(* IEC 61131-3 sources: RL_MAR/experiments/results/ablation/Ablation_no_role_config_deepseek-ai_DeepSeek-V3.2_20260603_074104 (part 2) *)

(* ---- med_49.st ---- *)
FUNCTION_BLOCK SmartHVACSystem
VAR_INPUT
    TemperatureSensor : REAL; (* Temperature sensor reading *)
    HumiditySensor : REAL; (* Humidity sensor reading *)
    Enable : BOOL := TRUE; (* System enable *)
    Reset : BOOL := FALSE; (* System reset *)
    ManualMode : BOOL := FALSE; (* Manual mode override *)
    ManualHVACMode : INT := 0; (* Manual HVAC mode: 0=Off, 1=Cooling, 2=Heating, 3=Ventilation *)
    ManualFanSpeed : INT := 0; (* Manual fan speed: 0=Off, 1=Low, 2=Medium, 3=High *)
END_VAR

VAR_OUTPUT
    HVACMode : INT := 0; (* HVAC operating mode: 0=Off, 1=Cooling, 2=Heating, 3=Ventilation *)
    HVACFanSpeed : INT := 0; (* Fan speed: 0=Off, 1=Low, 2=Medium, 3=High *)
    SystemActive : BOOL := FALSE; (* System active status *)
    Alarm : BOOL := FALSE; (* System alarm *)
END_VAR

VAR
    DesiredTemperature : REAL := 24.0; (* Desired temperature setting *)
    DesiredHumidity : REAL := 50.0; (* Desired humidity setting *)
    TemperatureThreshold : REAL := 1.0; (* Temperature tolerance threshold *)
    HumidityThreshold : REAL := 5.0; (* Humidity tolerance threshold *)

    AdjustedHumidity : REAL; (* Sanitized humidity input *)
    AdjustedTemperature : REAL; (* Sanitized temperature input *)

    NeedsVentilation : BOOL; (* Flag for ventilation requirement *)
    NeedsHeating : BOOL; (* Flag for heating requirement *)
    NeedsCooling : BOOL; (* Flag for cooling requirement *)

    TempSanitized : BOOL; (* Temperature sanitization status *)
    HumSanitized : BOOL; (* Humidity sanitization status *)

    ModeTimer : TON; (* Timer for mode changes *)
    FanTimer : TON; (* Timer for fan speed changes *)

    TempArray : ARRAY[1..10] OF REAL; (* Temperature history buffer *)
    HumArray : ARRAY[1..10] OF REAL; (* Humidity history buffer *)
    AvgTemperature : REAL; (* Average temperature *)
    AvgHumidity : REAL; (* Average humidity *)

    i : INT; (* Loop counter *)
    ArrayIndex : INT := 1; (* Current array index *)
    SampleCount : INT := 0; (* Number of samples collected *)
END_VAR

// Main execution logic
IF Reset THEN
    // Reset system
    HVACMode := 0;
    HVACFanSpeed := 0;
    SystemActive := FALSE;
    Alarm := FALSE;
    AdjustedHumidity := 0.0;
    AdjustedTemperature := 0.0;
    NeedsVentilation := FALSE;
    NeedsHeating := FALSE;
    NeedsCooling := FALSE;
    TempSanitized := FALSE;
    HumSanitized := FALSE;
    AvgTemperature := 0.0;
    AvgHumidity := 0.0;
    SampleCount := 0;
    ArrayIndex := 1;

    FOR i := 1 TO 10 DO
        TempArray[i] := 0.0;
        HumArray[i] := 0.0;
    END_FOR;

ELSIF Enable THEN
    SystemActive := TRUE;

    // 1. Input Sanitization
    // Sanitize humidity input
    IF HumiditySensor < 0.0 THEN
        AdjustedHumidity := 0.0;
        HumSanitized := TRUE;
    ELSIF HumiditySensor > 100.0 THEN
        AdjustedHumidity := 100.0;
        HumSanitized := TRUE;
    ELSE
        AdjustedHumidity := HumiditySensor;
        HumSanitized := TRUE;
    END_IF;

    // Sanitize temperature input
    IF TemperatureSensor < -50.0 THEN
        AdjustedTemperature := -50.0;
        TempSanitized := TRUE;
    ELSIF TemperatureSensor > 100.0 THEN
        AdjustedTemperature := 100.0;
        TempSanitized := TRUE;
    ELSE
        AdjustedTemperature := TemperatureSensor;
        TempSanitized := TRUE;
    END_IF;

    // Check for sensor alarm conditions
    Alarm := NOT (TempSanitized AND HumSanitized);

    // 2. Data averaging for stability
    TempArray[ArrayIndex] := AdjustedTemperature;
    HumArray[ArrayIndex] := AdjustedHumidity;

    ArrayIndex := ArrayIndex + 1;
    IF ArrayIndex > 10 THEN
        ArrayIndex := 1;
    END_IF;

    IF SampleCount < 10 THEN
        SampleCount := SampleCount + 1;
    END_IF;

    // Calculate averages
    AvgTemperature := 0.0;
    AvgHumidity := 0.0;
    FOR i := 1 TO SampleCount DO
        AvgTemperature := AvgTemperature + TempArray[i];
        AvgHumidity := AvgHumidity + HumArray[i];
    END_FOR;

    IF SampleCount > 0 THEN
        AvgTemperature := AvgTemperature / SampleCount;
        AvgHumidity := AvgHumidity / SampleCount;
    END_IF;

    // 3. Determine System Requirements using averaged values
    // Ventilation requirement
    IF AvgHumidity < (DesiredHumidity - HumidityThreshold) THEN
        NeedsVentilation := TRUE;
    ELSE
        NeedsVentilation := FALSE;
    END_IF;

    // Heating requirement
    IF AvgTemperature < (DesiredTemperature - TemperatureThreshold) THEN
        NeedsHeating := TRUE;
    ELSE
        NeedsHeating := FALSE;
    END_IF;

    // Cooling requirement
    IF AvgTemperature > (DesiredTemperature + TemperatureThreshold) THEN
        NeedsCooling := TRUE;
    ELSE
        NeedsCooling := FALSE;
    END_IF;

    // 4. Control Logic with prioritization
    IF ManualMode THEN
        // Manual mode override
        HVACMode := LIMIT(0, ManualHVACMode, 3);
        HVACFanSpeed := LIMIT(0, ManualFanSpeed, 3);
    ELSE
        // Automatic mode with prioritization
        IF NeedsHeating THEN
            HVACMode := 2; // Heating
            HVACFanSpeed := 3; // High
        ELSIF NeedsCooling THEN
            HVACMode := 1; // Cooling
            HVACFanSpeed := 3; // High
        ELSIF NeedsVentilation THEN
            HVACMode := 3; // Ventilation
            HVACFanSpeed := 3; // High
        ELSE
            HVACMode := 0; // Off
            HVACFanSpeed := 0; // Off
        END_IF;
    END_IF;

    // Apply timers for mode stability
    ModeTimer(IN := (HVACMode <> 0), PT := T#2S);
    FanTimer(IN := (HVACFanSpeed <> 0), PT := T#1S);

    // Ensure system only reports active when timers are done
    IF NOT ModeTimer.Q THEN
        HVACMode := 0;
    END_IF;

    IF NOT FanTimer.Q THEN
        HVACFanSpeed := 0;
    END_IF;

ELSE
    // System disabled
    SystemActive := FALSE;
    HVACMode := 0;
    HVACFanSpeed := 0;
    NeedsVentilation := FALSE;
    NeedsHeating := FALSE;
    NeedsCooling := FALSE;
END_IF;

END_FUNCTION_BLOCK

(* ---- med_50.st ---- *)
FUNCTION_BLOCK CarParkingSystem
VAR_INPUT
    NewCarSlot : INT; (* Input for new car arrival slot number *)
END_VAR
VAR_OUTPUT
    Elevator1Busy : BOOL; (* Elevator 1 status - busy or idle *)
    Elevator2Busy : BOOL; (* Elevator 2 status - busy or idle *)
    Elevator1Position : INT; (* Elevator 1 current position *)
    Elevator2Position : INT; (* Elevator 2 current position *)
END_VAR
VAR
    Elevator1Target : INT; (* Elevator 1 target floor *)
    Elevator2Target : INT; (* Elevator 2 target floor *)
    CarSlots : ARRAY[1..100] OF BOOL; (* Array to represent parking slots - TRUE if occupied *)
    bInitialized : BOOL := FALSE; (* Initialization flag *)
    i : INT; (* Loop index *)
    PendingRequests1 : ARRAY[1..50] OF BOOL; (* Pending requests for Elevator 1 *)
    PendingRequests2 : ARRAY[51..100] OF BOOL; (* Pending requests for Elevator 2 *)
    ScanIndex1 : INT := 1; (* Scanning index for Elevator 1 *)
    ScanIndex2 : INT := 51; (* Scanning index for Elevator 2 *)
END_VAR

(* Initialization - executed once *)
IF NOT bInitialized THEN
    Elevator1Busy := FALSE;
    Elevator2Busy := FALSE;
    Elevator1Position := 0;
    Elevator2Position := 0;
    Elevator1Target := 0;
    Elevator2Target := 0;

    (* Initialize all parking slots as empty *)
    FOR i := 1 TO 100 DO
        CarSlots[i] := FALSE;
    END_FOR;

    (* Initialize pending request arrays *)
    FOR i := 1 TO 50 DO
        PendingRequests1[i] := FALSE;
    END_FOR;

    FOR i := 51 TO 100 DO
        PendingRequests2[i] := FALSE;
    END_FOR;

    bInitialized := TRUE;
END_IF;

(* Process new car arrival if valid *)
IF (NewCarSlot >= 1) AND (NewCarSlot <= 100) THEN
    IF NOT CarSlots[NewCarSlot] THEN
        CarSlots[NewCarSlot] := TRUE;

        (* Store request in appropriate pending queue *)
        IF NewCarSlot <= 50 THEN
            PendingRequests1[NewCarSlot] := TRUE;
        ELSE
            PendingRequests2[NewCarSlot] := TRUE;
        END_IF;
    END_IF;
END_IF;

(* Control Elevator 1 movement *)
IF Elevator1Busy THEN
    IF Elevator1Position < Elevator1Target THEN
        Elevator1Position := Elevator1Position + 1;
    ELSIF Elevator1Position > Elevator1Target THEN
        Elevator1Position := Elevator1Position - 1;
    ELSE
        (* Elevator reached target - mark slot as serviced *)
        IF (Elevator1Target >= 1) AND (Elevator1Target <= 50) THEN
            PendingRequests1[Elevator1Target] := FALSE;
        END_IF;
        Elevator1Busy := FALSE;
    END_IF;
END_IF;

(* Control Elevator 2 movement *)
IF Elevator2Busy THEN
    IF Elevator2Position < Elevator2Target THEN
        Elevator2Position := Elevator2Position + 1;
    ELSIF Elevator2Position > Elevator2Target THEN
        Elevator2Position := Elevator2Position - 1;
    ELSE
        (* Elevator reached target - mark slot as serviced *)
        IF (Elevator2Target >= 51) AND (Elevator2Target <= 100) THEN
            PendingRequests2[Elevator2Target] := FALSE;
        END_IF;
        Elevator2Busy := FALSE;
    END_IF;
END_IF;

(* Idle elevator scanning for pending requests - Elevator 1 *)
IF NOT Elevator1Busy THEN
    (* Check for pending requests with round-robin scanning *)
    FOR i := 0 TO 49 DO
        ScanIndex1 := ScanIndex1 + 1;
        IF ScanIndex1 > 50 THEN
            ScanIndex1 := 1;
        END_IF;

        IF PendingRequests1[ScanIndex1] THEN
            Elevator1Target := ScanIndex1;
            Elevator1Busy := TRUE;
            EXIT;
        END_IF;
    END_FOR;
END_IF;

(* Idle elevator scanning for pending requests - Elevator 2 *)
IF NOT Elevator2Busy THEN
    (* Check for pending requests with round-robin scanning *)
    FOR i := 0 TO 49 DO
        ScanIndex2 := ScanIndex2 + 1;
        IF ScanIndex2 > 100 THEN
            ScanIndex2 := 51;
        END_IF;

        IF PendingRequests2[ScanIndex2] THEN
            Elevator2Target := ScanIndex2;
            Elevator2Busy := TRUE;
            EXIT;
        END_IF;
    END_FOR;
END_IF;

END_FUNCTION_BLOCK

(* ---- med_51.st ---- *)
FUNCTION_BLOCK PizzaMakingMachine
VAR_INPUT
    StartButton : BOOL;
    StopButton : BOOL;
    DoughReadySensor : BOOL;
    ToppingsReadySensor : BOOL;
    BakingDoneSensor : BOOL;
END_VAR

VAR_OUTPUT
    DoughRollerMotor : BOOL;
    ToppingDispenser : BOOL;
    ConveyorMotor : BOOL;
    OvenHeater : BOOL;
    OvenTemperature : INT;
END_VAR

VAR
    State : INT;
    OvenTargetTemp : INT;
END_VAR

// State definitions
CONSTANT
    STATE_IDLE : INT := 0;
    STATE_ROLLING_DOUGH : INT := 1;
    STATE_ADDING_TOPPINGS : INT := 2;
    STATE_MOVING_TO_OVEN : INT := 3;
    STATE_BAKING : INT := 4;
    STATE_COMPLETE : INT := 5;
END_CONSTANT

// Main state machine logic
IF StopButton THEN
    // Emergency stop - reset everything
    State := STATE_IDLE;
    DoughRollerMotor := FALSE;
    ToppingDispenser := FALSE;
    ConveyorMotor := FALSE;
    OvenHeater := FALSE;
    OvenTargetTemp := 0;
ELSE
    CASE State OF
        STATE_IDLE:
            DoughRollerMotor := FALSE;
            ToppingDispenser := FALSE;
            ConveyorMotor := FALSE;
            OvenHeater := FALSE;
            OvenTargetTemp := 0;

            IF StartButton THEN
                State := STATE_ROLLING_DOUGH;
            END_IF;

        STATE_ROLLING_DOUGH:
            DoughRollerMotor := TRUE;
            ToppingDispenser := FALSE;
            ConveyorMotor := FALSE;
            OvenHeater := FALSE;
            OvenTargetTemp := 0;

            IF DoughReadySensor THEN
                State := STATE_ADDING_TOPPINGS;
            END_IF;

        STATE_ADDING_TOPPINGS:
            DoughRollerMotor := FALSE;
            ToppingDispenser := TRUE;
            ConveyorMotor := FALSE;
            OvenHeater := FALSE;
            OvenTargetTemp := 0;

            IF ToppingsReadySensor THEN
                State := STATE_MOVING_TO_OVEN;
            END_IF;

        STATE_MOVING_TO_OVEN:
            DoughRollerMotor := FALSE;
            ToppingDispenser := FALSE;
            ConveyorMotor := TRUE;
            OvenHeater := TRUE; // Start heating oven
            OvenTargetTemp := 220;

            // Assume conveyor moves pizza to oven automatically
            // In real system, would have position sensor
            State := STATE_BAKING;

        STATE_BAKING:
            DoughRollerMotor := FALSE;
            ToppingDispenser := FALSE;
            ConveyorMotor := FALSE;
            OvenHeater := TRUE;
            OvenTargetTemp := 220;

            IF BakingDoneSensor THEN
                State := STATE_COMPLETE;
            END_IF;

        STATE_COMPLETE:
            DoughRollerMotor := FALSE;
            ToppingDispenser := FALSE;
            ConveyorMotor := FALSE;
            OvenHeater := FALSE;
            OvenTargetTemp := 0;

            // Wait for next start command
            IF NOT StartButton THEN
                State := STATE_IDLE;
            END_IF;

    END_CASE;
END_IF;

// Set oven temperature output
OvenTemperature := OvenTargetTemp;

END_FUNCTION_BLOCK

(* ---- med_52.st ---- *)
FUNCTION_BLOCK TrafficManagementSystem
VAR_INPUT
    VehicleCount1 : INT;
    VehicleCount2 : INT;
    VehicleCount3 : INT;
    VehicleCount4 : INT;
END_VAR

VAR_OUTPUT
    TrafficLight1 : BOOL;  (* TRUE = Green, FALSE = Red *)
    TrafficLight2 : BOOL;
    TrafficLight3 : BOOL;
    TrafficLight4 : BOOL;
END_VAR

VAR
    // Internal state variables for tie-breaking
    PrevPair1State : BOOL := TRUE;  (* Default to Intersection 1 green *)
    PrevPair2State : BOOL := TRUE;  (* Default to Intersection 3 green *)
END_VAR

(* Pair 1: Intersection 1 vs Intersection 2 *)
IF VehicleCount1 > VehicleCount2 THEN
    TrafficLight1 := TRUE;
    TrafficLight2 := FALSE;
    PrevPair1State := TRUE;
ELSIF VehicleCount2 > VehicleCount1 THEN
    TrafficLight1 := FALSE;
    TrafficLight2 := TRUE;
    PrevPair1State := FALSE;
ELSE
    (* Equal counts: use previous state to maintain complementary lights *)
    TrafficLight1 := PrevPair1State;
    TrafficLight2 := NOT PrevPair1State;
END_IF;

(* Pair 2: Intersection 3 vs Intersection 4 *)
IF VehicleCount3 > VehicleCount4 THEN
    TrafficLight3 := TRUE;
    TrafficLight4 := FALSE;
    PrevPair2State := TRUE;
ELSIF VehicleCount4 > VehicleCount3 THEN
    TrafficLight3 := FALSE;
    TrafficLight4 := TRUE;
    PrevPair2State := FALSE;
ELSE
    (* Equal counts: use previous state to maintain complementary lights *)
    TrafficLight3 := PrevPair2State;
    TrafficLight4 := NOT PrevPair2State;
END_IF;

END_FUNCTION_BLOCK

(* ---- med_53.st ---- *)
FUNCTION_BLOCK PouchMachine
VAR_INPUT
    start_machine: BOOL;
    stop_machine: BOOL;
END_VAR

VAR_OUTPUT
    machine_ready: BOOL;
    feeder_running: BOOL;
    cutter_running: BOOL;
    heating_running: BOOL;
    cooling_running: BOOL;
END_VAR

VAR
    startup_complete: BOOL := FALSE;
    shutdown_complete: BOOL := FALSE;
    current_state: INT := 0;
    next_state: INT := 0;

    // Timers for state transitions
    heating_timer: TON;
    cooling_timer: TON;
    feeder_timer: TON;
    cutter_timer: TON;

    // Additional internal variables
    tension_established: BOOL;
    heating_stations_active: ARRAY[1..8] OF BOOL;
    cooling_stations_active: ARRAY[1..8] OF BOOL;
    horizontal_cutter_active: BOOL;
    vertical_cutter_active: BOOL;
    feeder1_active: BOOL;
    feeder2_active: BOOL;

    // Loop counter
    i: INT;
END_VAR

// Initialize timers with preset times
heating_timer(IN := FALSE, PT := T#2S);
cooling_timer(IN := FALSE, PT := T#2S);
feeder_timer(IN := FALSE, PT := T#3S);
cutter_timer(IN := FALSE, PT := T#1S);

CASE current_state OF
    0: (* Idle State *)
        machine_ready := FALSE;
        feeder_running := FALSE;
        cutter_running := FALSE;
        heating_running := FALSE;
        cooling_running := FALSE;
        startup_complete := FALSE;
        shutdown_complete := FALSE;
        tension_established := FALSE;

        // Reset all stations
        FOR i := 1 TO 8 DO
            heating_stations_active[i] := FALSE;
            cooling_stations_active[i] := FALSE;
        END_FOR;

        horizontal_cutter_active := FALSE;
        vertical_cutter_active := FALSE;
        feeder1_active := FALSE;
        feeder2_active := FALSE;

        // Reset all timers
        heating_timer(IN := FALSE);
        cooling_timer(IN := FALSE);
        feeder_timer(IN := FALSE);
        cutter_timer(IN := FALSE);

        // Transition to start sequence
        IF start_machine AND NOT stop_machine THEN
            next_state := 1;
        ELSE
            next_state := 0;
        END_IF;

    1: (* Start Heating Stations *)
        heating_running := TRUE;

        // Activate all 8 heating stations
        FOR i := 1 TO 8 DO
            heating_stations_active[i] := TRUE;
        END_FOR;

        // Start timer for heating stabilization
        heating_timer(IN := TRUE);
        IF heating_timer.Q THEN
            next_state := 2;
            heating_timer(IN := FALSE);
        ELSE
            next_state := 1;
        END_IF;

    2: (* Start Cooling Stations *)
        cooling_running := TRUE;

        // Activate all 8 cooling stations
        FOR i := 1 TO 8 DO
            cooling_stations_active[i] := TRUE;
        END_FOR;

        // Start timer for cooling stabilization
        cooling_timer(IN := TRUE);
        IF cooling_timer.Q THEN
            next_state := 3;
            cooling_timer(IN := FALSE);
        ELSE
            next_state := 2;
        END_IF;

    3: (* Start Feeders with Tension Control *)
        feeder_running := TRUE;
        feeder1_active := TRUE;
        feeder2_active := TRUE;

        // Start timer for tension establishment
        feeder_timer(IN := TRUE);
        IF feeder_timer.Q THEN
            // Tension established after timer expires
            tension_established := TRUE;
            next_state := 4;
            feeder_timer(IN := FALSE);
        ELSE
            tension_established := FALSE;
            next_state := 3;
        END_IF;

    4: (* Start Cutters *)
        cutter_running := TRUE;
        horizontal_cutter_active := TRUE;
        vertical_cutter_active := TRUE;

        // Start timer for cutter activation
        cutter_timer(IN := TRUE);
        IF cutter_timer.Q THEN
            next_state := 5;
            cutter_timer(IN := FALSE);
        ELSE
            next_state := 4;
        END_IF;

    5: (* Machine Ready *)
        machine_ready := TRUE;
        startup_complete := TRUE;

        // Wait for stop command
        IF stop_machine THEN
            next_state := 6;
        ELSE
            next_state := 5;
        END_IF;

    6: (* Stop Cutters *)
        cutter_running := FALSE;
        horizontal_cutter_active := FALSE;
        vertical_cutter_active := FALSE;

        // Start timer for cutter deactivation
        cutter_timer(IN := TRUE);
        IF cutter_timer.Q THEN
            next_state := 7;
            cutter_timer(IN := FALSE);
        ELSE
            next_state := 6;
        END_IF;

    7: (* Stop Feeders *)
        feeder_running := FALSE;
        feeder1_active := FALSE;
        feeder2_active := FALSE;
        tension_established := FALSE;

        // Start timer for feeder shutdown
        feeder_timer(IN := TRUE);
        IF feeder_timer.Q THEN
            next_state := 8;
            feeder_timer(IN := FALSE);
        ELSE
            next_state := 7;
        END_IF;

    8: (* Stop Cooling Stations *)
        cooling_running := FALSE;

        // Deactivate all 8 cooling stations
        FOR i := 1 TO 8 DO
            cooling_stations_active[i] := FALSE;
        END_FOR;

        // Start timer for cooling shutdown
        cooling_timer(IN := TRUE);
        IF cooling_timer.Q THEN
            next_state := 9;
            cooling_timer(IN := FALSE);
        ELSE
            next_state := 8;
        END_IF;

    9: (* Stop Heating Stations *)
        heating_running := FALSE;

        // Deactivate all 8 heating stations
        FOR i := 1 TO 8 DO
            heating_stations_active[i] := FALSE;
        END_FOR;

        // Start timer for heating shutdown
        heating_timer(IN := TRUE);
        IF heating_timer.Q THEN
            next_state := 10;
            heating_timer(IN := FALSE);
        ELSE
            next_state := 9;
        END_IF;

    10: (* Shutdown Complete *)
        machine_ready := FALSE;
        shutdown_complete := TRUE;

        // Return to idle when stop signal is released
        IF NOT stop_machine THEN
            next_state := 0;
        ELSE
            next_state := 10;
        END_IF;

    ELSE
        // Safety fallback to idle state
        next_state := 0;
END_CASE;

// Update state for next scan cycle
current_state := next_state;

END_FUNCTION_BLOCK

(* ---- med_54.st ---- *)
FUNCTION_BLOCK FeedForwardControl
VAR_INPUT
    FlowRate1, FlowRate2: REAL; // Input flow rates of reactants
    MixRatio: REAL; // Desired mixing ratio (Reactant1:Reactant2)
END_VAR

VAR_OUTPUT
    OutFlowRate1, OutFlowRate2: REAL; // Output flow rates for reactants to maintain the mixing ratio
END_VAR

VAR
    MixedFlowRate: REAL; // Total mixed flow rate
    TempFlowRate1: REAL;
    TempFlowRate2: REAL;
    LimitedFlowRate1: REAL;
    LimitedFlowRate2: REAL;
END_VAR

// 1. VALIDATE AND LIMIT INPUT FLOW RATES (0 to 100)
IF FlowRate1 < 0.0 THEN
    LimitedFlowRate1 := 0.0;
ELSIF FlowRate1 > 100.0 THEN
    LimitedFlowRate1 := 100.0;
ELSE
    LimitedFlowRate1 := FlowRate1;
END_IF;

IF FlowRate2 < 0.0 THEN
    LimitedFlowRate2 := 0.0;
ELSIF FlowRate2 > 100.0 THEN
    LimitedFlowRate2 := 100.0;
ELSE
    LimitedFlowRate2 := FlowRate2;
END_IF;

// 2. CALCULATE TOTAL MIXED FLOW RATE
MixedFlowRate := LimitedFlowRate1 + LimitedFlowRate2;

// 3. CALCULATE OUTPUT FLOW RATES WITH ERROR HANDLING
IF MixRatio = 0.0 THEN
    // Prevent division by zero - use equal distribution
    TempFlowRate1 := MixedFlowRate / 2.0;
    TempFlowRate2 := MixedFlowRate / 2.0;
ELSE
    // Calculate based on mixing ratio: MixRatio = Reactant1:Reactant2
    // For ratio a:b, Reactant1 fraction = a/(a+b)
    TempFlowRate1 := MixedFlowRate * (MixRatio / (MixRatio + 1.0));
    TempFlowRate2 := MixedFlowRate * (1.0 / (MixRatio + 1.0));
END_IF;

// 4. LIMIT OUTPUT FLOW RATES TO ALLOWED RANGE (0 to 100)
IF TempFlowRate1 < 0.0 THEN
    OutFlowRate1 := 0.0;
ELSIF TempFlowRate1 > 100.0 THEN
    OutFlowRate1 := 100.0;
ELSE
    OutFlowRate1 := TempFlowRate1;
END_IF;

IF TempFlowRate2 < 0.0 THEN
    OutFlowRate2 := 0.0;
ELSIF TempFlowRate2 > 100.0 THEN
    OutFlowRate2 := 100.0;
ELSE
    OutFlowRate2 := TempFlowRate2;
END_IF;

// 5. ENSURE OUTPUT CONSISTENCY (Optional safeguard)
// Additional check to ensure outputs don't exceed total mixed flow rate
IF (OutFlowRate1 + OutFlowRate2) > MixedFlowRate THEN
    // Scale down proportionally if needed
    TempFlowRate1 := OutFlowRate1;
    TempFlowRate2 := OutFlowRate2;
    OutFlowRate1 := TempFlowRate1 * (MixedFlowRate / (TempFlowRate1 + TempFlowRate2));
    OutFlowRate2 := TempFlowRate2 * (MixedFlowRate / (TempFlowRate1 + TempFlowRate2));
END_IF;

END_FUNCTION_BLOCK

(* ---- med_55.st ---- *)
FUNCTION_BLOCK StateMachineControl
VAR_INPUT
    request : BOOL;
    done : BOOL;
END_VAR

VAR_OUTPUT
    listen : BOOL;
END_VAR

VAR
    state : INT := 0;
END_VAR

(* State machine logic *)
CASE state OF
    0: (* Idle state *)
        listen := TRUE;
        IF request THEN
            state := 1; (* Transition to Processing *)
            listen := FALSE;
        END_IF;

    1: (* Processing state *)
        listen := FALSE;
        IF done THEN
            state := 0; (* Transition to Idle *)
        END_IF;

    ELSE
        (* Error recovery - reset to Idle state *)
        state := 0;
        listen := TRUE;
END_CASE;

END_FUNCTION_BLOCK

(* ---- med_56.st ---- *)
FUNCTION_BLOCK FB_SimpleRepeat
VAR_INPUT
    INPUT_VAR1 : INT := 2;
    INPUT_COUNTER : INT := 4;
END_VAR

VAR_OUTPUT
    OUTPUT_VAR1 : INT;
END_VAR

VAR
    COUNTER : INT;
END_VAR

METHOD Main : BOOL
VAR_INPUT
    Execute : BOOL;
END_VAR
VAR_OUTPUT
    Done : BOOL;
END_VAR

    IF Execute THEN
        OUTPUT_VAR1 := INPUT_VAR1;
        COUNTER := INPUT_COUNTER;

        REPEAT
            OUTPUT_VAR1 := OUTPUT_VAR1 * 2;
            COUNTER := COUNTER - 1;
        UNTIL COUNTER <= 0
        END_REPEAT;

        Done := TRUE;
    ELSE
        Done := FALSE;
    END_IF;

    Main := Done;
END_METHOD

END_FUNCTION_BLOCK

(* ---- med_57.st ---- *)
FUNCTION_BLOCK FB_CourseDifferenceControl
VAR_INPUT
    KOMPASS_GRAD : INT;
    KURS : INT;
END_VAR
VAR_OUTPUT
    KURS_DIFF : INT;
END_VAR
VAR
    diff_temp : INT;
END_VAR

// Main logic
IF KOMPASS_GRAD < 0 THEN
    KURS_DIFF := 0;
ELSE
    diff_temp := KURS - KOMPASS_GRAD;

    // Apply range correction for angles
    IF diff_temp > 1800 THEN
        diff_temp := diff_temp - 3600;
    ELSIF diff_temp < -1800 THEN
        diff_temp := diff_temp + 3600;
    END_IF;

    KURS_DIFF := diff_temp;
END_IF;
END_FUNCTION_BLOCK

PROGRAM MAIN
VAR
    fbCourseDiff : FB_CourseDifferenceControl;
    kompass_grad_input : INT;
    kurs_input : INT;
    kurs_diff_output : INT;
END_VAR

// Call the function block
fbCourseDiff(KOMPASS_GRAD := kompass_grad_input, KURS := kurs_input);
kurs_diff_output := fbCourseDiff.KURS_DIFF;
END_PROGRAM

(* ---- med_58.st ---- *)
FUNCTION_BLOCK FB_ThresholdAccumulator
VAR_INPUT
    i : INT;
END_VAR

VAR_OUTPUT
    o : INT;
END_VAR

VAR
    s1 : INT;
END_VAR

// Initialize s1 to 0 at the start of each function block call
s1 := 0;

// If the input i is greater than 0, add its value to s1
IF i > 0 THEN
    s1 := s1 + i;
END_IF;

// After the first condition, if s1 equals 42, add 8000 to s1
IF s1 = 42 THEN
    s1 := s1 + 8000;
END_IF;

// Determine final output
IF s1 < 0 THEN
    o := 0;
ELSE
    o := s1;
END_IF;

END_FUNCTION_BLOCK

(* ---- med_59.st ---- *)
FUNCTION_BLOCK FB_ConditionalSelectAndAggregate
VAR_INPUT
    Z : INT;
END_VAR
VAR
    A_X : INT := 42;
    A_Y : INT := 333;
END_VAR
VAR_OUTPUT
    NEW_Z : INT;
END_VAR

IF A_X > Z THEN
    NEW_Z := A_Y;
ELSE
    NEW_Z := Z;
END_IF;
NEW_Z := NEW_Z + A_X + A_Y;
END_FUNCTION_BLOCK

(* ---- med_60.st ---- *)
FUNCTION_BLOCK FB_RequestHandler
VAR_INPUT
    request : BOOL;
    done : BOOL;
END_VAR

VAR_OUTPUT
    listen : BOOL;
END_VAR

VAR
    currentState : INT := 0;
    nextState : INT := 0;
END_VAR

CASE currentState OF
    0: (* State 0 - Idle/Listening *)
        listen := TRUE;

        IF request THEN
            listen := FALSE;
            nextState := 1;
        ELSE
            nextState := 0;
        END_IF;

    1: (* State 1 - Processing *)
        listen := FALSE;

        IF done THEN
            listen := TRUE;
            nextState := 0;
        ELSE
            nextState := 1;
        END_IF;

    ELSE
        (* Default case - return to state 0 if invalid state *)
        currentState := 0;
        nextState := 0;
        listen := TRUE;
END_CASE;

currentState := nextState;
END_FUNCTION_BLOCK

(* ---- med_61.st ---- *)
FUNCTION_BLOCK FB_Sum
VAR_INPUT
    maxValue : INT;
END_VAR
VAR_OUTPUT
    wData : WORD;
END_VAR
VAR
    II : INT;
    tempSum : DINT;
END_VAR

tempSum := 0;
FOR II := 0 TO maxValue DO
    tempSum := tempSum + II;
END_FOR;
wData := WORD(tempSum);
END_FUNCTION_BLOCK

(* ---- med_62.st ---- *)
FUNCTION_BLOCK FB_PedestrianTrafficLight
VAR_INPUT
    pedBtnPress : BOOL;
END_VAR
VAR_OUTPUT
    carLightIsGreen : BOOL;
    pedLightIsGreen : BOOL;
    counter : INT;
END_VAR
VAR
    buttonPressedBefore : BOOL := FALSE;
    state : INT := 1; // 1: Normal, 2: Wait for ped green, 3: Ped green, 4: Wait for car green
END_VAR

// State machine logic
CASE state OF
    1: // Normal state - Car green, Ped red
        carLightIsGreen := TRUE;
        pedLightIsGreen := FALSE;
        counter := 0;

        // Detect rising edge of button press
        IF pedBtnPress AND NOT buttonPressedBefore THEN
            state := 2;
        END_IF;

    2: // Car red, waiting for pedestrian green
        carLightIsGreen := FALSE;
        pedLightIsGreen := FALSE;
        counter := counter + 1;

        IF counter >= 10 THEN
            state := 3;
        END_IF;

    3: // Car red, pedestrian green
        carLightIsGreen := FALSE;
        pedLightIsGreen := TRUE;
        counter := counter + 1;

        IF counter >= 40 THEN
            state := 4;
        END_IF;

    4: // Car red, waiting for car green
        carLightIsGreen := FALSE;
        pedLightIsGreen := FALSE;
        counter := counter + 1;

        IF counter >= 50 THEN
            state := 1;
        END_IF;
END_CASE;

// Update button press tracking
buttonPressedBefore := pedBtnPress;

END_FUNCTION_BLOCK

(* ---- med_63.st ---- *)
FUNCTION MoveCarToExitGate : BOOL
VAR_INPUT
    SpaceNumber : INT;
END_VAR
// Car movement logic implementation
// Return TRUE when movement is successfully completed
MoveCarToExitGate := TRUE;
END_FUNCTION

FUNCTION_BLOCK Automated_Parking_Controller
VAR_INPUT
    EntryGateSensor : BOOL; (* Sensor input for entry gate *)
    ExitGateSensor : BOOL; (* Sensor input for exit gate *)
    CarDetected : BOOL; (* Sensor input for car detection *)
END_VAR
VAR_OUTPUT
    ParkingSpaceNumber : INT := 0; (* Allocated parking space number *)
    RetrievalInProgress : BOOL := FALSE; (* Flag for car retrieval in progress *)
END_VAR
VAR
    ParkingSpaces : ARRAY[1..100] OF BOOL; (* Parking space status: TRUE=Occupied, FALSE=Available *)
    i : INT; (* Loop counter *)
    AssignedSpace : INT := 0; (* Temporary storage for assigned space *)
    RetrievalComplete : BOOL := FALSE; (* Flag to track retrieval completion *)
END_VAR

// Entry Gate Management
IF EntryGateSensor AND NOT RetrievalInProgress THEN
    // Find first available parking space
    AssignedSpace := 0;
    FOR i := 1 TO 100 DO
        IF NOT ParkingSpaces[i] AND AssignedSpace = 0 THEN
            ParkingSpaces[i] := TRUE; // Mark as occupied
            ParkingSpaceNumber := i; // Output assigned space number
            AssignedSpace := i;
        END_IF
    END_FOR;
END_IF;

// Exit Gate Management
IF ExitGateSensor AND ParkingSpaceNumber > 0 THEN
    // Mark the corresponding parking space as available
    ParkingSpaces[ParkingSpaceNumber] := FALSE;
    ParkingSpaceNumber := 0; // Reset output
END_IF;

// Car Retrieval Management
IF CarDetected AND NOT RetrievalInProgress AND ParkingSpaceNumber > 0 THEN
    RetrievalInProgress := TRUE;
    RetrievalComplete := FALSE;
END_IF;

IF RetrievalInProgress THEN
    // Execute retrieval logic
    RetrievalComplete := MoveCarToExitGate(ParkingSpaceNumber);

    IF RetrievalComplete THEN
        // Mark parking space as available
        ParkingSpaces[ParkingSpaceNumber] := FALSE;
        ParkingSpaceNumber := 0; // Reset output
        RetrievalInProgress := FALSE; // Reset flag
    END_IF;
END_IF;
END_FUNCTION_BLOCK

(* ---- med_64.st ---- *)
FUNCTION_BLOCK BakeryOvenControl
VAR_INPUT
    TemperatureSensor : REAL;           (* Current oven temperature reading *)
    HumiditySensor : REAL;              (* Current oven humidity reading *)
    StartOven : BOOL;                   (* Command to start the oven *)
    TemperatureSetpoint : REAL;         (* Desired temperature setpoint *)
    HumiditySetpoint : REAL;            (* Desired humidity setpoint *)
    BakingTimeSetpoint : TIME;          (* Total baking time *)
    TemperatureThreshold : REAL := 2.0; (* Temperature control deadband *)
    HumidityThreshold : REAL := 5.0;    (* Humidity control deadband *)
END_VAR

VAR_OUTPUT
    HeatingElement : BOOL;              (* Control signal for heating element *)
    CoolingElement : BOOL;              (* Control signal for cooling element *)
    HumidityControl : BOOL;             (* Control signal for humidification *)
    DehumidityControl : BOOL;           (* Control signal for dehumidification *)
    OvenActive : BOOL;                  (* Oven status: TRUE when baking *)
    RemainingTime : TIME;               (* Remaining baking time *)
END_VAR

VAR
    BakingTimer : TON;                  (* Timer for baking duration *)
    OneSecondPulse : TON;               (* Timer for 1-second pulse generation *)
    PulseSignal : BOOL;                 (* Internal 1-second pulse *)
    InternalRemainingTime : TIME;       (* Internal remaining time counter *)
END_VAR

(* Initialize timers *)
OneSecondPulse(IN := NOT OneSecondPulse.Q, PT := T#1S);
PulseSignal := OneSecondPulse.Q;

(* Oven control logic *)
IF StartOven AND NOT OvenActive THEN
    (* Start baking cycle *)
    OvenActive := TRUE;
    InternalRemainingTime := BakingTimeSetpoint;
    BakingTimer(IN := TRUE, PT := BakingTimeSetpoint);
ELSIF NOT StartOven THEN
    (* Manual stop or initialization *)
    OvenActive := FALSE;
    BakingTimer(IN := FALSE, PT := T#0S);
END_IF

(* Decrement remaining time when oven is active *)
IF OvenActive AND PulseSignal THEN
    IF InternalRemainingTime >= T#1S THEN
        InternalRemainingTime := InternalRemainingTime - T#1S;
    ELSE
        InternalRemainingTime := T#0S;
    END_IF;
END_IF;

(* Stop oven when timer expires *)
IF BakingTimer.Q THEN
    OvenActive := FALSE;
END_IF;

(* Temperature control - only active when oven is on *)
IF OvenActive THEN
    HeatingElement := TemperatureSensor < (TemperatureSetpoint - TemperatureThreshold);
    CoolingElement := TemperatureSensor > (TemperatureSetpoint + TemperatureThreshold);
ELSE
    HeatingElement := FALSE;
    CoolingElement := FALSE;
END_IF;

(* Humidity control - only active when oven is on *)
IF OvenActive THEN
    HumidityControl := HumiditySensor < (HumiditySetpoint - HumidityThreshold);
    DehumidityControl := HumiditySensor > (HumiditySetpoint + HumidityThreshold);
ELSE
    HumidityControl := FALSE;
    DehumidityControl := FALSE;
END_IF;

(* Output remaining time *)
RemainingTime := InternalRemainingTime;

(* Ensure all outputs are off when oven is not active *)
IF NOT OvenActive THEN
    HeatingElement := FALSE;
    CoolingElement := FALSE;
    HumidityControl := FALSE;
    DehumidityControl := FALSE;
    InternalRemainingTime := T#0S;
END_IF;
END_FUNCTION_BLOCK

(* ---- med_65.st ---- *)
FUNCTION_BLOCK TheaterControl
VAR_INPUT
    StartButton : BOOL;        (* Input for starting a performance *)
    StopButton : BOOL;         (* Input for stopping a performance *)
    SceneNumber : INT;         (* Input for selecting the scene or act *)
END_VAR
VAR_OUTPUT
    LightingControl : BOOL;    (* Output for controlling lighting *)
    SoundControl : BOOL;       (* Output for controlling sound *)
    PerformanceInProgress : BOOL; (* Indicator for an ongoing performance *)
END_VAR
VAR
    bStartRisingEdge : BOOL;
    bStopRisingEdge : BOOL;
    bPrevStart : BOOL := FALSE;
    bPrevStop : BOOL := FALSE;
END_VAR

(* Detect rising edges for button presses *)
bStartRisingEdge := StartButton AND NOT bPrevStart;
bStopRisingEdge := StopButton AND NOT bPrevStop;
bPrevStart := StartButton;
bPrevStop := StopButton;

(* Main control logic with stop button having highest priority *)
IF bStopRisingEdge THEN
    (* Immediate stop - override all other inputs *)
    LightingControl := FALSE;
    SoundControl := FALSE;
    PerformanceInProgress := FALSE;
ELSIF bStartRisingEdge AND NOT PerformanceInProgress THEN
    (* Start performance only if not already in progress *)
    IF (SceneNumber >= 1) AND (SceneNumber <= 3) THEN
        (* Valid scene - activate outputs *)
        LightingControl := TRUE;
        SoundControl := TRUE;
        PerformanceInProgress := TRUE;
    ELSE
        (* Invalid scene - keep outputs inactive *)
        LightingControl := FALSE;
        SoundControl := FALSE;
        PerformanceInProgress := FALSE;
    END_IF;
END_IF;

(* Note: Outputs maintain their state until changed by the logic above *)
END_FUNCTION_BLOCK

(* ---- med_66.st ---- *)
FUNCTION_BLOCK ElevatorControl
VAR_INPUT
    CurrentPos : INT;
    RequestedPos : INT;
    ButtonPressed : BOOL;
END_VAR
VAR_OUTPUT
    MotorMovingUp : BOOL;
    MotorMovingDown : BOOL;
    DoorIsOpen : BOOL;
END_VAR
VAR
    bMoving : BOOL := FALSE;
END_VAR

// Main elevator control logic
IF ButtonPressed THEN
    // Start movement when button is pressed
    bMoving := TRUE;
    DoorIsOpen := FALSE;
END_IF;

IF bMoving THEN
    // Elevator is in motion
    IF RequestedPos > CurrentPos THEN
        // Move upward
        MotorMovingUp := TRUE;
        MotorMovingDown := FALSE;
        DoorIsOpen := FALSE;
    ELSIF RequestedPos < CurrentPos THEN
        // Move downward
        MotorMovingUp := FALSE;
        MotorMovingDown := TRUE;
        DoorIsOpen := FALSE;
    ELSE
        // Reached target floor
        MotorMovingUp := FALSE;
        MotorMovingDown := FALSE;
        DoorIsOpen := TRUE;
        bMoving := FALSE;
    END_IF;
ELSE
    // Elevator is stationary
    MotorMovingUp := FALSE;
    MotorMovingDown := FALSE;

    // Keep door open if at requested position, otherwise closed
    IF CurrentPos = RequestedPos THEN
        DoorIsOpen := TRUE;
    ELSE
        DoorIsOpen := FALSE;
    END_IF;
END_IF;

END_FUNCTION_BLOCK

(* ---- med_67.st ---- *)
FUNCTION_BLOCK FB_FactorialCalculator
VAR_INPUT
    X : INT;
END_VAR

VAR_OUTPUT
    FactorialResult : INT;
    FactorialGoodResult : INT;
END_VAR

VAR
END_VAR

// Initialize outputs
FactorialGoodResult := 0;
FactorialResult := 0;

// Check if input is within safe range
IF (X >= -3) AND (X <= 3) THEN
    // Calculate X^4 (X multiplied by itself 4 times)
    FactorialGoodResult := X * X * X * X;

    // Calculate FactorialResult based on FactorialGoodResult
    IF FactorialGoodResult > 1 THEN
        FactorialResult := FactorialGoodResult * (FactorialGoodResult - 1);
    ELSE
        FactorialResult := FactorialGoodResult;
    END_IF;
ELSE
    // Overflow prevention for inputs outside range
    FactorialResult := 1;
    FactorialGoodResult := 0;
END_IF;

END_FUNCTION_BLOCK

(* ---- med_68.st ---- *)
FUNCTION_BLOCK SignalControl
VAR_INPUT
    Int1 : BOOL;
    Int2 : BOOL;
    Int3 : BOOL;
    Int4 : BOOL;
    Int5 : BOOL;
    Int6 : BOOL;
    Int7 : BOOL;
    Int8 : BOOL;
    IntAn1 : UINT;
    IntAn2 : UINT;
    IntAn3 : UINT;
    IntAn4 : UINT;
    IntAn5 : UINT;
    IntAn6 : UINT;
    IntAn7 : UINT;
    IntAn8 : UINT;
    Marca2 : BOOL;
END_VAR

VAR_OUTPUT
    Out1 : BOOL;
    Out2 : BOOL;
    Out3 : BOOL;
    Out4 : BOOL;
    Out5 : BOOL;
    Out6 : BOOL;
    Out7 : BOOL;
    Out8 : BOOL;
    OutAn1 : UINT;
    OutAn2 : UINT;
    OutAn3 : UINT;
    OutAn4 : UINT;
    OutAn5 : UINT;
    OutAn6 : UINT;
    OutAn7 : UINT;
    OutAn8 : UINT;
END_VAR

VAR
    Marca1 : BOOL;
END_VAR

// Main logic execution
// Logic for Marca1 flag
IF NOT Marca2 AND (Marca1 OR NOT Out1) AND Int1 THEN
    Marca1 := TRUE;
ELSE
    Marca1 := FALSE;
END_IF;

// Logic for Marca2 flag (note: Marca2 is both input and internal state)
IF NOT Marca1 AND (Marca2 OR Out1) AND Int1 THEN
    Marca2 := TRUE;
ELSE
    Marca2 := FALSE;
END_IF;

// Latch behavior for Out1
IF NOT Marca2 AND (Marca1 OR Out1) THEN
    Out1 := TRUE;
ELSE
    Out1 := FALSE;
END_IF;

// Boolean pass-through for Out2, Out3, Out4
Out2 := Int2;
Out3 := Int3;
Out4 := Int4;

// Unsigned integer pass-through for OutAn1 to OutAn4
OutAn1 := IntAn1;
OutAn2 := IntAn2;
OutAn3 := IntAn3;
OutAn4 := IntAn4;

// Conditional output logic for Out5 to Out8
// Out5 condition: IntAn5 > 1000 AND NOT Int5
Out5 := (IntAn5 > 1000) AND NOT Int5;

// Out6 condition: IntAn6 > 1000 AND NOT Int6
Out6 := (IntAn6 > 1000) AND NOT Int6;

// Out7 condition: IntAn7 > 1000 AND NOT Int7
Out7 := (IntAn7 > 1000) AND NOT Int7;

// Out8 condition: IntAn8 > 1000 AND NOT Int8
Out8 := (IntAn8 > 1000) AND NOT Int8;

// Pass-through for analog outputs OutAn5 to OutAn8
OutAn5 := IntAn5;
OutAn6 := IntAn6;
OutAn7 := IntAn7;
OutAn8 := IntAn8;

END_FUNCTION_BLOCK

(* ---- med_69.st ---- *)
FUNCTION_BLOCK FB_ValueOut
VAR_INPUT
    valueIn : INT;
    conf : UINT;
END_VAR
VAR_OUTPUT
    ValueOut : INT;
END_VAR

CASE conf OF
    1,2:
        ValueOut := valueIn / 10;

    3:
        IF valueIn = 0 THEN
            ValueOut := 0;
        ELSIF valueIn = 300 THEN
            ValueOut := 163;
        ELSIF valueIn = 600 THEN
            ValueOut := 331;
        ELSE
            ValueOut := 0;
        END_IF;

    6,7:
        IF valueIn = 100 THEN
            ValueOut := 319;
        ELSE
            ValueOut := 0;
        END_IF;

    ELSE
        ValueOut := 0;
END_CASE;

END_FUNCTION_BLOCK

(* ---- med_70.st ---- *)
FUNCTION_BLOCK EggIncubatorControl
VAR_INPUT
    StartButton : BOOL;          (* Input for starting the incubation process *)
    StopButton : BOOL;           (* Input for stopping the incubation process *)
    TemperatureSensor : REAL;    (* Input for temperature reading in °C *)
    HumiditySensor : REAL;       (* Input for humidity reading in % *)
END_VAR
VAR_OUTPUT
    HeatingElement : BOOL;       (* Output for controlling the heating element *)
    Humidifier : BOOL;           (* Output for controlling the humidifier *)
    EggTurningMotor : BOOL;      (* Output for controlling the egg turning motor *)
    IncubationInProgress : BOOL; (* Indicator for an ongoing incubation process *)
END_VAR
VAR
    TargetTemperature : REAL;    (* Target temperature in °C *)
    TargetHumidity : REAL;       (* Target humidity in % *)
    TurnIntervalSeconds : INT;   (* Interval for turning eggs (1 hour in seconds) *)
    TurnTimerSeconds : INT;      (* Timer for egg turning cycle in seconds *)
END_VAR

(* Initialize control parameters *)
TargetTemperature := 37.5;
TargetHumidity := 50.0;
TurnIntervalSeconds := 3600;

(* Start/Stop Control *)
IF StopButton THEN
    IncubationInProgress := FALSE;
    HeatingElement := FALSE;
    Humidifier := FALSE;
    EggTurningMotor := FALSE;
    TurnTimerSeconds := 0;
ELSIF StartButton AND NOT IncubationInProgress THEN
    IncubationInProgress := TRUE;
END_IF;

(* Temperature Control *)
IF IncubationInProgress THEN
    IF TemperatureSensor < TargetTemperature THEN
        HeatingElement := TRUE;
    ELSE
        HeatingElement := FALSE;
    END_IF;
ELSE
    HeatingElement := FALSE;
END_IF;

(* Humidity Control *)
IF IncubationInProgress THEN
    IF HumiditySensor < TargetHumidity THEN
        Humidifier := TRUE;
    ELSE
        Humidifier := FALSE;
    END_IF;
ELSE
    Humidifier := FALSE;
END_IF;

(* Egg Turning Cycle *)
IF IncubationInProgress THEN
    TurnTimerSeconds := TurnTimerSeconds + 1;
    IF TurnTimerSeconds >= TurnIntervalSeconds THEN
        EggTurningMotor := NOT EggTurningMotor;
        TurnTimerSeconds := 0;
    END_IF;
ELSE
    TurnTimerSeconds := 0;
END_IF;

END_FUNCTION_BLOCK

(* ---- med_71.st ---- *)
FUNCTION_BLOCK FB_Fibonacci_Calculator
VAR_INPUT
    N : DINT := 5;
END_VAR
VAR_OUTPUT
    O : DINT := 1;
END_VAR
VAR
    F1 : DINT := 1;
    F2 : DINT := 1;
    CNT : DINT := 2;
    TempSum : DINT;
END_VAR

(* Handle edge cases: N <= 2 returns 1 *)
IF N <= 2 THEN
    O := 1;
ELSE
    (* Initialize Fibonacci sequence *)
    F1 := 1;
    F2 := 1;
    CNT := 2;

    (* Calculate Fibonacci numbers up to N-th term *)
    WHILE CNT < N DO
        TempSum := F1 + F2;

        (* Apply saturation arithmetic: clamp at INT maximum (32767) *)
        IF TempSum > 32767 THEN
            F2 := 32767;
            EXIT;  (* Exit loop early when saturation limit reached *)
        END_IF;

        (* Update Fibonacci values for next iteration *)
        F1 := F2;
        F2 := TempSum;
        CNT := CNT + 1;
    END_WHILE;

    (* Set output to the N-th Fibonacci number *)
    O := F2;
END_IF;
END_FUNCTION_BLOCK

(* ---- med_72.st ---- *)
FUNCTION_BLOCK DigitalSignageManagement
VAR_INPUT
    DisplayLocations : ARRAY[1..10] OF BOOL;    (* Display active status per location *)
    ContentSource : ARRAY[1..10] OF INT;        (* Requested content per location *)
END_VAR
VAR_OUTPUT
    CurrentContent : ARRAY[1..10] OF INT;       (* Actual displayed content per location *)
END_VAR
VAR
    i : INT;                                    (* Loop index *)
END_VAR

(* Process all 10 display locations *)
FOR i := 1 TO 10 DO
    IF DisplayLocations[i] THEN
        (* Display is active - validate content code *)
        CASE ContentSource[i] OF
            1: CurrentContent[i] := 1;          (* News *)
            2: CurrentContent[i] := 2;          (* Weather *)
            3: CurrentContent[i] := 3;          (* Promotional Content *)
        ELSE
            CurrentContent[i] := 0;             (* Invalid code - show no content *)
        END_CASE;
    ELSE
        (* Display is inactive - always show no content *)
        CurrentContent[i] := 0;
    END_IF;
END_FOR;

END_FUNCTION_BLOCK

(* ---- med_73.st ---- *)
FUNCTION_BLOCK RoboticWeldingSystem
VAR_INPUT
    RobotArm1Ready : BOOL;    (* Input for robot arm 1 ready status *)
    RobotArm2Ready : BOOL;    (* Input for robot arm 2 ready status *)
    WeldingGunReady : BOOL;   (* Input for welding gun ready status *)
    StartButton : BOOL;       (* Input for start button press *)
    StopButton : BOOL;        (* Input for stop button press *)
END_VAR
VAR_OUTPUT
    WeldingTrigger : BOOL;    (* Output to trigger welding *)
    WeldingComplete : BOOL;   (* Output indicating welding completion *)
END_VAR
VAR
    bAllReady : BOOL;         (* Internal flag for all components ready *)
END_VAR

(* Check if all components are ready *)
bAllReady := RobotArm1Ready AND RobotArm2Ready AND WeldingGunReady;

(* Main safety logic with stop button having highest priority *)
IF StopButton THEN
    (* Immediate stop when stop button is pressed *)
    WeldingTrigger := FALSE;
    WeldingComplete := TRUE;
ELSIF bAllReady AND StartButton THEN
    (* Start welding only when all components ready AND start button pressed *)
    WeldingTrigger := TRUE;
    WeldingComplete := FALSE;
ELSE
    (* Default state - no welding *)
    WeldingTrigger := FALSE;
    WeldingComplete := TRUE;
END_IF;

END_FUNCTION_BLOCK

(* ---- med_74.st ---- *)
FUNCTION_BLOCK TrafficManagementSystem
VAR_INPUT
    VehicleCount1 : INT; (* Vehicle count at intersection 1 *)
    VehicleCount2 : INT; (* Vehicle count at intersection 2 *)
    VehicleCount3 : INT; (* Vehicle count at intersection 3 *)
    VehicleCount4 : INT; (* Vehicle count at intersection 4 *)
END_VAR

VAR_OUTPUT
    TrafficLight1 : BOOL; (* TRUE = Green, FALSE = Red *)
    TrafficLight2 : BOOL; (* TRUE = Green, FALSE = Red *)
    TrafficLight3 : BOOL; (* TRUE = Green, FALSE = Red *)
    TrafficLight4 : BOOL; (* TRUE = Green, FALSE = Red *)
END_VAR

VAR
    (* Internal state variables for clarity *)
    TrafficLightState1 : BOOL;
    TrafficLightState2 : BOOL;
    TrafficLightState3 : BOOL;
    TrafficLightState4 : BOOL;
END_VAR

(* Control logic for intersection pair 1 (Intersection 1 and 2) *)
IF VehicleCount1 > VehicleCount2 THEN
    TrafficLightState1 := TRUE;   (* Green for intersection 1 *)
    TrafficLightState2 := FALSE;  (* Red for intersection 2 *)
ELSIF VehicleCount1 < VehicleCount2 THEN
    TrafficLightState1 := FALSE;  (* Red for intersection 1 *)
    TrafficLightState2 := TRUE;   (* Green for intersection 2 *)
ELSE
    (* Equal counts: both red for safety *)
    TrafficLightState1 := FALSE;
    TrafficLightState2 := FALSE;
END_IF;

(* Control logic for intersection pair 2 (Intersection 3 and 4) *)
IF VehicleCount3 > VehicleCount4 THEN
    TrafficLightState3 := TRUE;   (* Green for intersection 3 *)
    TrafficLightState4 := FALSE;  (* Red for intersection 4 *)
ELSIF VehicleCount3 < VehicleCount4 THEN
    TrafficLightState3 := FALSE;  (* Red for intersection 3 *)
    TrafficLightState4 := TRUE;   (* Green for intersection 4 *)
ELSE
    (* Equal counts: both red for safety *)
    TrafficLightState3 := FALSE;
    TrafficLightState4 := FALSE;
END_IF;

(* Assign internal states to outputs *)
TrafficLight1 := TrafficLightState1;
TrafficLight2 := TrafficLightState2;
TrafficLight3 := TrafficLightState3;
TrafficLight4 := TrafficLightState4;

END_FUNCTION_BLOCK

(* ---- med_75.st ---- *)
FUNCTION_BLOCK HomeBrewingSystem
VAR_INPUT
    TemperatureSensor : REAL; (* Input for temperature measurement (°C) *)
    WaterFlowSensor : REAL; (* Input for water flow measurement (L/min) *)
    BrewingStartTime : TIME; (* Input for brewing process start time *)
    BrewingDuration : TIME; (* Input for total brewing duration *)
END_VAR

VAR_OUTPUT
    HeatingElement : BOOL; (* Output to control heating element *)
    AgitationMotor : BOOL; (* Output to control agitation motor *)
    HopsDispenser : BOOL; (* Output to control hops dispenser *)
    FermentationTank : BOOL; (* Output to control fermentation tank *)
END_VAR

VAR
    ElapsedBrewingTime : TIME; (* Time elapsed since brewing start *)
    HopsDispensed : BOOL; (* Flag to track if hops have been dispensed *)
    TankTransferred : BOOL; (* Flag to track if transfer to fermentation tank has occurred *)
    CurrentTime : TIME; (* Current system time *)
    HopsTime : TIME := T#5h; (* Time threshold for hops dispensing *)
    FermentationTime : TIME := T#48h; (* Time threshold for fermentation transfer *)
    TargetTemperature : REAL := 65.0; (* Target brewing temperature *)
    FlowThreshold : REAL := 0.5; (* Flow threshold for agitation motor *)
END_VAR

(* Main program logic *)
CurrentTime := TIME(); (* Get current system time *)

(* Calculate elapsed brewing time *)
IF BrewingStartTime > T#0s THEN
    ElapsedBrewingTime := CurrentTime - BrewingStartTime;

    (* Ensure elapsed time doesn't exceed brewing duration *)
    IF ElapsedBrewingTime > BrewingDuration THEN
        ElapsedBrewingTime := BrewingDuration;
    END_IF;
ELSE
    ElapsedBrewingTime := T#0s;
END_IF;

(* Temperature control logic *)
HeatingElement := TemperatureSensor < TargetTemperature;

(* Agitation motor control logic *)
AgitationMotor := WaterFlowSensor > FlowThreshold;

(* Hops dispensing logic - activate after 5 hours, only once *)
IF (ElapsedBrewingTime >= HopsTime) AND (NOT HopsDispensed) AND (ElapsedBrewingTime <= BrewingDuration) THEN
    HopsDispenser := TRUE;
    HopsDispensed := TRUE;
ELSE
    HopsDispenser := FALSE;
END_IF;

(* Fermentation tank transfer logic - activate after 48 hours, only once *)
IF (ElapsedBrewingTime >= FermentationTime) AND (NOT TankTransferred) AND (ElapsedBrewingTime <= BrewingDuration) THEN
    FermentationTank := TRUE;
    TankTransferred := TRUE;
ELSE
    FermentationTank := FALSE;
END_IF;

(* Reset flags when brewing duration is complete or not started *)
IF (ElapsedBrewingTime >= BrewingDuration) OR (BrewingStartTime = T#0s) THEN
    HopsDispensed := FALSE;
    TankTransferred := FALSE;
END_IF;

END_FUNCTION_BLOCK

(* ---- med_76.st ---- *)
FUNCTION_BLOCK MultimediaArtInstallationControl
VAR_INPUT
    MotionSensor : BOOL;           (* Motion detection input *)
    AudioTrack : BOOL;             (* Selected audio track *)
    VisualContent : BOOL;          (* Selected visual content *)
END_VAR

VAR_OUTPUT
    LightingControl : BOOL;        (* Lighting control output *)
    AudioControl : BOOL;           (* Audio playback control *)
    VisualControl : BOOL;          (* Visual display control *)
    ActivationTime : TIME;         (* Activation duration *)
END_VAR

VAR
    ActivationTimer : TON;         (* Timer for activation duration *)
    TimerPreset : TIME := T#300S;  (* Predefined limit: 300 seconds *)
    PreviousMotion : BOOL;         (* Edge detection for motion *)
    bMotionDetected : BOOL;        (* Internal motion detection flag *)
END_VAR

(* Initialize timer *)
ActivationTimer(IN := bMotionDetected, PT := TimerPreset);

(* Motion detection with edge detection *)
IF MotionSensor AND NOT PreviousMotion THEN
    bMotionDetected := TRUE;
ELSIF NOT MotionSensor THEN
    bMotionDetected := FALSE;
END_IF;
PreviousMotion := MotionSensor;

(* Control multimedia elements based on motion detection *)
LightingControl := bMotionDetected;
AudioControl := bMotionDetected AND AudioTrack;
VisualControl := bMotionDetected AND VisualContent;

(* Update activation time output *)
ActivationTime := ActivationTimer.ET;

(* Safety protocol: Deactivate all elements and reset timer if no motion *)
IF NOT bMotionDetected THEN
    ActivationTimer(IN := FALSE, PT := TimerPreset);
END_IF;

(* Additional safety check: Ensure elements are off when timer reaches preset *)
IF ActivationTimer.Q THEN
    bMotionDetected := FALSE;
    ActivationTimer(IN := FALSE, PT := TimerPreset);
END_IF;
END_FUNCTION_BLOCK

(* ---- med_77.st ---- *)
FUNCTION_BLOCK OutdoorLEDLightingControl
VAR_INPUT
    AmbientLight : REAL;    (* Ambient light sensor input in Lux *)
    MotionSensor : BOOL;    (* Motion sensor input (TRUE = motion detected) *)
    EnergySaving : BOOL;    (* Energy saving mode input (TRUE = energy saving ON) *)
END_VAR

VAR_OUTPUT
    Light : BOOL;           (* LED lighting control output (TRUE = lights ON) *)
    EnergyMode : BOOL;      (* Energy saving mode status output *)
END_VAR

(* Main control logic *)
IF MotionSensor THEN
    (* Motion detection override *)
    Light := TRUE;
    EnergyMode := FALSE;
ELSE
    (* No motion detected - apply ambient light and energy saving logic *)
    IF (AmbientLight < 50.0) AND (NOT EnergySaving) THEN
        Light := TRUE;
    ELSE
        Light := FALSE;
    END_IF;

    (* Energy mode always reflects the EnergySaving input *)
    EnergyMode := EnergySaving;
END_IF;

END_FUNCTION_BLOCK

(* ---- med_78.st ---- *)
FUNCTION_BLOCK RetractableRoofControl
VAR_INPUT
    RainSensor : BOOL;           (* TRUE if rain is detected *)
    WindSensor : BOOL;           (* TRUE if strong wind is detected *)
    TemperatureSensor : REAL;    (* Current temperature in degrees *)
END_VAR
VAR_OUTPUT
    RoofMotor : BOOL;            (* TRUE closes roof, FALSE opens roof *)
END_VAR
VAR
    bCombinedCondition : BOOL;
    bRainOnlyCondition : BOOL;
    bLowTempCondition : BOOL;
END_VAR

(* Evaluate conditions *)
bCombinedCondition := RainSensor AND WindSensor;
bRainOnlyCondition := RainSensor AND NOT bCombinedCondition;
bLowTempCondition := (TemperatureSensor < 20.0) AND NOT bCombinedCondition AND NOT bRainOnlyCondition;

(* Priority-based control logic *)
IF bCombinedCondition THEN
    (* Highest priority: both rain and strong wind *)
    RoofMotor := TRUE;
ELSIF bRainOnlyCondition THEN
    (* Second priority: rain only *)
    RoofMotor := TRUE;
ELSIF bLowTempCondition THEN
    (* Third priority: low temperature *)
    RoofMotor := TRUE;
ELSE
    (* Normal conditions: open roof *)
    RoofMotor := FALSE;
END_IF;

END_FUNCTION_BLOCK

(* ---- med_79.st ---- *)
FUNCTION_BLOCK CapsuleFillingMachineControl
VAR_INPUT
    CapsuleWeight : REAL;           (* Current capsule weight *)
    TargetWeight : REAL;            (* Target weight to achieve *)
    CapsuleInPosition : BOOL;       (* Capsule position sensor *)
    HopperEmpty : BOOL;             (* Hopper empty sensor *)
    HopperLowSensor : BOOL;         (* Hopper low level sensor *)
END_VAR
VAR_OUTPUT
    FeederMotor : BOOL;             (* Feeder motor control *)
    FillingMotor : BOOL;            (* Filling motor control *)
    ConveyorMotor : BOOL;           (* Conveyor motor control *)
    FillingInProgress : BOOL;       (* Filling status *)
    ErrorFlag : BOOL;               (* General error flag *)
    ErrorCode : INT;                (* Error code: 0=OK, 1=Capsule not detected, 2=Filling timeout *)
    HopperLowWarning : BOOL;        (* Hopper low level warning *)
END_VAR
VAR
    (* State machine *)
    State : INT := 0;               (* 0=IDLE, 1=CONVEYING, 2=FILLING, 3=CONVEYING_OUT, 4=ERROR *)

    (* Timers *)
    ConveyingTimer : TON;           (* Timer for conveying capsule to position *)
    FillingTimer : TON;             (* Timer for filling operation *)
    ConveyOutTimer : TON;           (* Timer for conveying filled capsule out *)
    CapsuleDetectTimer : TON;       (* Timer for capsule detection timeout *)
    FillingTimeoutTimer : TON;      (* Timer for filling timeout *)

    (* Control parameters *)
    Tolerance : REAL := 0.02;       (* Weight tolerance as percentage of target *)
    ConveyingTime : TIME := T#2S;   (* Time to convey capsule to position *)
    ConveyOutTime : TIME := T#1S;   (* Time to convey capsule out *)
    CapsuleDetectTimeout : TIME := T#5S; (* Timeout for capsule detection *)
    FillingTimeout : TIME := T#10S; (* Timeout for filling operation *)

    (* Internal flags *)
    CapsuleDetected : BOOL;         (* Capsule detected flag *)
    FillingComplete : BOOL;         (* Filling completion flag *)
    WeightTolerance : REAL;         (* Calculated weight tolerance *)

    (* Edge detection *)
    PrevCapsuleInPosition : BOOL;   (* Previous state of capsule sensor *)

    (* Filling control *)
    FastFillThreshold : REAL := 0.7; (* Threshold for fast/slow filling (70% of target) *)
    FillingSpeed : REAL;            (* Calculated filling speed *)
    MaxFillingSpeed : REAL := 100.0; (* Maximum filling speed *)
    MinFillingSpeed : REAL := 20.0; (* Minimum filling speed for trickle feed *)
END_VAR

(* Calculate weight tolerance *)
WeightTolerance := TargetWeight * Tolerance;

(* Hopper low level warning *)
HopperLowWarning := HopperLowSensor;

(* Safety Check: Hopper Empty *)
IF HopperEmpty THEN
    FeederMotor := FALSE;
    FillingMotor := FALSE;
    ConveyorMotor := FALSE;
    FillingInProgress := FALSE;
    State := 0;  (* Return to IDLE state *)
    RETURN;
END_IF;

(* Weight Validation: Initial Check *)
IF CapsuleWeight >= (TargetWeight - WeightTolerance) THEN
    FeederMotor := FALSE;
    FillingMotor := FALSE;
    ConveyorMotor := FALSE;
    FillingInProgress := FALSE;
    State := 0;  (* Return to IDLE state *)
    RETURN;
END_IF;

(* Main state machine *)
CASE State OF
    (* State 0: IDLE *)
    0:
        (* Reset all outputs *)
        FillingMotor := FALSE;
        ConveyorMotor := FALSE;
        FillingInProgress := FALSE;
        ErrorFlag := FALSE;
        ErrorCode := 0;

        (* Control feeder motor based on hopper level *)
        FeederMotor := NOT HopperLowSensor;

        (* Reset internal flags *)
        CapsuleDetected := FALSE;
        FillingComplete := FALSE;

        (* Reset timers *)
        ConveyingTimer(IN := FALSE, PT := ConveyingTime);
        FillingTimer(IN := FALSE, PT := FillingTimeout);
        ConveyOutTimer(IN := FALSE, PT := ConveyOutTime);
        CapsuleDetectTimer(IN := FALSE, PT := CapsuleDetectTimeout);
        FillingTimeoutTimer(IN := FALSE, PT := FillingTimeout);

        (* Transition to CONVEYING when capsule is detected *)
        IF CapsuleInPosition AND NOT PrevCapsuleInPosition THEN
            CapsuleDetected := TRUE;
            State := 1;  (* Move to CONVEYING state *)
        END_IF;

    (* State 1: CONVEYING *)
    1:
        FillingInProgress := FALSE;
        ConveyorMotor := TRUE;
        FeederMotor := NOT HopperLowSensor;

        (* Start conveying timer *)
        ConveyingTimer(IN := TRUE, PT := ConveyingTime);

        (* Start capsule detection timeout timer *)
        CapsuleDetectTimer(IN := TRUE, PT := CapsuleDetectTimeout);

        (* Check for capsule detection timeout *)
        IF CapsuleDetectTimer.Q THEN
            ErrorFlag := TRUE;
            ErrorCode := 1;  (* Capsule not detected error *)
            State := 4;      (* Move to ERROR state *)
        END_IF;

        (* Transition to FILLING when conveying time elapsed *)
        IF ConveyingTimer.Q THEN
            ConveyorMotor := FALSE;
            State := 2;  (* Move to FILLING state *)
        END_IF;

    (* State 2: FILLING *)
    2:
        FillingInProgress := TRUE;
        ConveyorMotor := FALSE;
        FeederMotor := NOT HopperLowSensor;

        (* Start filling timeout timer *)
        FillingTimeoutTimer(IN := TRUE, PT := FillingTimeout);

        (* Advanced filling control with fast/slow phases *)
        IF CapsuleWeight < (TargetWeight * FastFillThreshold) THEN
            (* Fast filling phase *)
            FillingSpeed := MaxFillingSpeed;
            FillingMotor := TRUE;
        ELSE
            (* Slow trickle feed phase *)
            FillingSpeed := MinFillingSpeed;

            (* Calculate remaining weight difference *)
            IF (TargetWeight - CapsuleWeight) > WeightTolerance THEN
                FillingMotor := TRUE;
            ELSE
                FillingMotor := FALSE;
                FillingComplete := TRUE;
            END_IF;
        END_IF;

        (* Check for filling completion *)
        IF CapsuleWeight >= (TargetWeight - WeightTolerance) THEN
            FillingMotor := FALSE;
            FillingComplete := TRUE;
            State := 3;  (* Move to CONVEYING_OUT state *)
        END_IF;

        (* Check for filling timeout *)
        IF FillingTimeoutTimer.Q THEN
            ErrorFlag := TRUE;
            ErrorCode := 2;  (* Filling timeout error *)
            State := 4;      (* Move to ERROR state *)
        END_IF;

    (* State 3: CONVEYING_OUT *)
    3:
        FillingInProgress := FALSE;
        FillingMotor := FALSE;
        ConveyorMotor := TRUE;
        FeederMotor := NOT HopperLowSensor;

        (* Start convey out timer *)
        ConveyOutTimer(IN := TRUE, PT := ConveyOutTime);

        (* Transition back to IDLE when convey out time elapsed *)
        IF ConveyOutTimer.Q THEN
            ConveyorMotor := FALSE;
            State := 0;  (* Return to IDLE state *)
        END_IF;

    (* State 4: ERROR *)
    4:
        (* Safety stop all motors *)
        FeederMotor := FALSE;
        FillingMotor := FALSE;
        ConveyorMotor := FALSE;
        FillingInProgress := FALSE;

        (* Error state persists until manually reset *)
        (* To reset: Set State := 0 from external program *)

END_CASE;

(* Update edge detection variable *)
PrevCapsuleInPosition := CapsuleInPosition;

END_FUNCTION_BLOCK

(* ---- med_80.st ---- *)
FUNCTION_BLOCK DoughMixerControl
VAR_INPUT
    IngredientsDetected : BOOL;
END_VAR
VAR_OUTPUT
    MixingInProgress : BOOL;
END_VAR
VAR
    MixingTimeElapsed : TIME;
    MixingTimeLimit : TIME := T#5S;
    PrevIngredientsDetected : BOOL;
END_VAR

(* Rising edge detection for ingredient presence *)
IF IngredientsDetected AND NOT PrevIngredientsDetected THEN
    (* Start mixing cycle *)
    MixingInProgress := TRUE;
    MixingTimeElapsed := T#0S;
ELSIF NOT IngredientsDetected OR MixingTimeElapsed >= MixingTimeLimit THEN
    (* Stop conditions: ingredients removed or time limit reached *)
    MixingInProgress := FALSE;
END_IF;

(* Increment timer while mixing is active *)
IF MixingInProgress THEN
    MixingTimeElapsed := MixingTimeElapsed + T#1S;
END_IF;

(* Store current state for edge detection in next cycle *)
PrevIngredientsDetected := IngredientsDetected;
END_FUNCTION_BLOCK

(* ---- med_81.st ---- *)
FUNCTION_BLOCK SolarPanelTracking
VAR_INPUT
    CurrentTime : TIME;
    SolarIntensity : REAL;
END_VAR

VAR_OUTPUT
    PanelAngle : REAL;
END_VAR

VAR
    SunriseTime : TIME := T#6H;
    NoonTime : TIME := T#12H;
    SunsetTime : TIME := T#18H;
    MorningAngle : REAL := 30.0;
    NoonAngle : REAL := 60.0;
    EveningAngle : REAL := 30.0;
END_VAR

// Main logic
IF SolarIntensity >= 90.0 THEN
    // Solar intensity override - highest priority
    PanelAngle := NoonAngle;
ELSE
    // Time-based tracking
    IF (CurrentTime < SunriseTime) OR (CurrentTime >= SunsetTime) THEN
        // Nighttime
        PanelAngle := 0.0;
    ELSIF (CurrentTime >= SunriseTime) AND (CurrentTime < NoonTime) THEN
        // Morning period
        PanelAngle := MorningAngle;
    ELSIF (CurrentTime >= NoonTime) AND (CurrentTime < SunsetTime) THEN
        // Afternoon/Evening period
        PanelAngle := EveningAngle;
    ELSE
        // Fallback (should not occur with proper time ranges)
        PanelAngle := 0.0;
    END_IF;
END_IF;

END_FUNCTION_BLOCK

(* ---- med_82.st ---- *)
FUNCTION_BLOCK PetFeederControl
VAR_INPUT
    CurrentTime : TIME; (* Current system time from RTC *)
END_VAR

VAR_OUTPUT
    FoodDispense : BOOL; (* Food dispenser control signal *)
END_VAR

VAR
    FeedTime1 : TIME := T#8H0M0S; (* First feeding time - 8:00 AM *)
    FeedTime2 : TIME := T#12H0M0S; (* Second feeding time - 12:00 PM *)
    FeedTime3 : TIME := T#18H0M0S; (* Third feeding time - 6:00 PM *)
    FoodAmount : INT := 50; (* Reserved for future use - currently unused *)
END_VAR

(* Main logic implementation *)
FoodDispense := FALSE;

IF (CurrentTime >= FeedTime1) AND (CurrentTime < FeedTime1 + T#30S) THEN
    FoodDispense := TRUE;
ELSIF (CurrentTime >= FeedTime2) AND (CurrentTime < FeedTime2 + T#30S) THEN
    FoodDispense := TRUE;
ELSIF (CurrentTime >= FeedTime3) AND (CurrentTime < FeedTime3 + T#30S) THEN
    FoodDispense := TRUE;
END_IF;

END_FUNCTION_BLOCK

(* ---- med_83.st ---- *)
FUNCTION_BLOCK AmusementRideControl
VAR_INPUT
    StartButton : BOOL;     (* Start button input *)
    StopButton : BOOL;      (* Emergency stop button input *)
    SpeedSensor : REAL;     (* Speed sensor input (RPM) *)
    SafetySensor : BOOL;    (* Safety sensor status *)
END_VAR
VAR_OUTPUT
    MotorOn : BOOL := FALSE;    (* Motor control output *)
    BrakeOn : BOOL := TRUE;     (* Brake control output *)
END_VAR
VAR
    SpeedLimit : REAL := 60.0;  (* Maximum allowed speed in RPM *)
END_VAR

(* Main safety control logic *)
IF StopButton THEN
    (* Emergency Stop - Highest Priority *)
    MotorOn := FALSE;
    BrakeOn := TRUE;
ELSIF StartButton AND (NOT StopButton) AND (SpeedSensor <= SpeedLimit) AND SafetySensor THEN
    (* Start Condition - All conditions must be met *)
    MotorOn := TRUE;
    BrakeOn := FALSE;
ELSE
    (* Default/Fail-Safe State *)
    MotorOn := FALSE;
    BrakeOn := TRUE;
END_IF;

(* Continuous monitoring during normal operation *)
IF MotorOn THEN
    IF (SpeedSensor > SpeedLimit) OR (NOT SafetySensor) THEN
        (* Safety violation during operation *)
        MotorOn := FALSE;
        BrakeOn := TRUE;
    END_IF;
END_IF;

END_FUNCTION_BLOCK

(* ---- med_84.st ---- *)
FUNCTION_BLOCK ParcelSortingSystem
VAR_INPUT
    ParcelSizeSensor : REAL;     (* Sensor input for parcel size in millimeters *)
    DestinationCodeSensor : INT; (* Destination code: 1=Location A, 2=Location B *)
END_VAR

VAR_OUTPUT
    ConveyorBeltMotor : BOOL;    (* Output for conveyor belt motor: TRUE=On, FALSE=Off *)
    SortingGate1 : BOOL;         (* Output for sorting gate 1: TRUE=Open, FALSE=Closed *)
    SortingGate2 : BOOL;         (* Output for sorting gate 2: TRUE=Open, FALSE=Closed *)
END_VAR

VAR
    bSizeValid : BOOL;           (* Flag indicating valid parcel size *)
    bDestValid : BOOL;           (* Flag indicating valid destination code *)
    bIsLargeParcel : BOOL;       (* Flag indicating large parcel *)
    bIsSmallParcel : BOOL;       (* Flag indicating small parcel *)
    bDestLocationA : BOOL;       (* Flag for destination Location A *)
    bDestLocationB : BOOL;       (* Flag for destination Location B *)

    (* Constants for size thresholds *)
    LARGE_SIZE_THRESHOLD : REAL := 500.0;  (* Parcels >= 500mm are considered large *)
    MIN_VALID_SIZE : REAL := 50.0;         (* Minimum valid parcel size *)
    MAX_VALID_SIZE : REAL := 1000.0;       (* Maximum valid parcel size *)
END_VAR

(* Main program logic *)
METHOD ProcessParcelSorting
    (* Initialize all outputs to safe state *)
    ConveyorBeltMotor := FALSE;
    SortingGate1 := FALSE;
    SortingGate2 := FALSE;

    (* Validate parcel size *)
    bSizeValid := (ParcelSizeSensor >= MIN_VALID_SIZE) AND
                  (ParcelSizeSensor <= MAX_VALID_SIZE);

    (* Validate destination code *)
    bDestValid := (DestinationCodeSensor = 1) OR (DestinationCodeSensor = 2);

    (* Determine parcel size category *)
    bIsLargeParcel := ParcelSizeSensor >= LARGE_SIZE_THRESHOLD;
    bIsSmallParcel := (ParcelSizeSensor < LARGE_SIZE_THRESHOLD) AND bSizeValid;

    (* Determine destination *)
    bDestLocationA := (DestinationCodeSensor = 1) AND bDestValid;
    bDestLocationB := (DestinationCodeSensor = 2) AND bDestValid;

    (* Main sorting logic *)
    IF bSizeValid AND bDestValid THEN
        (* Valid parcel detected - start conveyor *)
        ConveyorBeltMotor := TRUE;

        IF bIsLargeParcel THEN
            (* Large parcels always go to sorting gate 1 *)
            SortingGate1 := TRUE;
            SortingGate2 := FALSE;

        ELSIF bIsSmallParcel THEN
            (* Small parcels routing based on destination *)
            IF bDestLocationA THEN
                (* Small parcels for Location A go to sorting gate 2 *)
                SortingGate1 := FALSE;
                SortingGate2 := TRUE;
            ELSIF bDestLocationB THEN
                (* Small parcels for Location B stay on conveyor *)
                SortingGate1 := FALSE;
                SortingGate2 := FALSE;
            END_IF;
        END_IF;

    ELSE
        (* Invalid input detected - stop system and close all gates *)
        ConveyorBeltMotor := FALSE;
        SortingGate1 := FALSE;
        SortingGate2 := FALSE;
    END_IF;
END_METHOD
END_FUNCTION_BLOCK

(* ---- med_85.st ---- *)
FUNCTION_BLOCK ShredderControl
VAR_INPUT
    StartButton : BOOL;        (* Input for the start button *)
    StopButton : BOOL;         (* Input for the stop button *)
    EmergencyStop : BOOL;      (* Input for the emergency stop button *)
    MotorStatus : BOOL;        (* Feedback status of the shredder motor *)
    MaterialInFeed : BOOL;     (* Input for material being fed into the shredder *)
    JammedSensor : BOOL;       (* Input for detecting material jamming *)
END_VAR
VAR_OUTPUT
    MotorControl : BOOL;       (* Output for controlling the shredder motor *)
    SafetyRelay : BOOL;        (* Output for safety relay: TRUE=Safe, FALSE=Unsafe *)
END_VAR
VAR
    bMotorRunCmd : BOOL;       (* Internal motor run command *)
    bEmergencyCondition : BOOL; (* Combined emergency condition *)
END_VAR

(* Check for highest priority emergency conditions *)
bEmergencyCondition := EmergencyStop OR JammedSensor;

IF bEmergencyCondition THEN
    (* Emergency stop or jam detected - immediate shutdown *)
    bMotorRunCmd := FALSE;
    SafetyRelay := FALSE;
    MotorControl := FALSE;
ELSE
    (* Normal operation logic *)

    (* Start conditions: start button OR material feed (with no stop command) *)
    IF StartButton OR (MaterialInFeed AND NOT StopButton) THEN
        bMotorRunCmd := TRUE;
    END_IF;

    (* Stop condition: stop button *)
    IF StopButton THEN
        bMotorRunCmd := FALSE;
    END_IF;

    (* Safety relay active during normal operation *)
    SafetyRelay := TRUE;

    (* Control motor based on run command *)
    MotorControl := bMotorRunCmd;
END_IF;

END_FUNCTION_BLOCK

(* ---- med_86.st ---- *)
FUNCTION_BLOCK FruitJuicingBottling
VAR_INPUT
    StartButton : BOOL;        (* Input for starting the process *)
    StopButton : BOOL;         (* Input for stopping the process *)
    FruitSelected : BOOL;      (* Input indicating fruit selection *)
END_VAR
VAR_OUTPUT
    JuiceProcessing : BOOL;    (* Output for controlling juice extraction *)
    BottleFilling : BOOL;      (* Output for controlling bottle filling *)
    CapPlacement : BOOL;       (* Output for placing caps on bottles *)
    Packaging : BOOL;          (* Output for packaging filled bottles *)
    ProcessInProgress : BOOL;  (* Indicator for an ongoing process *)
END_VAR
VAR
    bProcessActive : BOOL;     (* Internal process state *)
END_VAR

(* Start condition: StartButton pressed, fruit selected, and no process running *)
IF StartButton AND FruitSelected AND NOT ProcessInProgress THEN
    bProcessActive := TRUE;
END_IF;

(* Stop condition: StopButton pressed OR fruit deselected during operation *)
IF StopButton OR NOT FruitSelected THEN
    bProcessActive := FALSE;
END_IF;

(* Process tracking output *)
ProcessInProgress := bProcessActive;

(* Concurrent process stages - all active when process is running *)
JuiceProcessing := ProcessInProgress;
BottleFilling := ProcessInProgress;
CapPlacement := ProcessInProgress;
Packaging := ProcessInProgress;

END_FUNCTION_BLOCK

(* ---- med_87.st ---- *)
FUNCTION_BLOCK WaterDesalination
VAR_INPUT
    StartButton : BOOL;           (* Input for starting the desalination process *)
    StopButton : BOOL;            (* Input for stopping the desalination process *)
    SalinitySensor : REAL;        (* Input for salinity level measurement *)
END_VAR
VAR_OUTPUT
    SeawaterInletValve : BOOL;    (* Output for seawater inlet valve control *)
    FreshwaterOutletValve : BOOL; (* Output for freshwater outlet valve control *)
    DesalinationInProgress : BOOL;(* Indicator for an ongoing desalination process *)
END_VAR
VAR
    MaxSalinity : REAL := 35.0;   (* Maximum allowable salinity in ppm for freshwater *)
    SalinityControlSeconds : INT := 0; (* Timer for salinity control in seconds *)
END_VAR

(* Start/Stop Control Logic *)
IF StopButton THEN
    (* Immediate stop when StopButton is pressed *)
    SeawaterInletValve := FALSE;
    FreshwaterOutletValve := FALSE;
    DesalinationInProgress := FALSE;
    SalinityControlSeconds := 0;
ELSIF StartButton AND NOT DesalinationInProgress THEN
    (* Start process when StartButton is pressed and process isn't already running *)
    SeawaterInletValve := TRUE;
    FreshwaterOutletValve := TRUE;
    DesalinationInProgress := TRUE;
END_IF;

(* Salinity Monitoring and Control Logic *)
IF DesalinationInProgress THEN
    (* Increment timer each cycle (assuming 1 second cycle time) *)
    SalinityControlSeconds := SalinityControlSeconds + 1;

    (* Check salinity every 10 seconds *)
    IF SalinityControlSeconds >= 10 THEN
        IF SalinitySensor > MaxSalinity THEN
            (* Close freshwater valve if salinity is too high *)
            FreshwaterOutletValve := FALSE;
        ELSE
            (* Keep freshwater valve open if salinity is acceptable *)
            FreshwaterOutletValve := TRUE;
        END_IF;
        (* Reset timer after check *)
        SalinityControlSeconds := 0;
    END_IF;
END_IF;

END_FUNCTION_BLOCK

(* ---- med_88.st ---- *)
FUNCTION_BLOCK SmartLockerControl
VAR_INPUT
    AccessCode : INT;     (* User entered access code *)
    LockerNumber : INT;   (* Selected locker number (1-10) *)
END_VAR
VAR_OUTPUT
    LockerOpen : BOOL;    (* TRUE when locker should open *)
END_VAR
VAR
    LockerStatus : ARRAY[1..10] OF BOOL := [TRUE,TRUE,TRUE,TRUE,TRUE,TRUE,TRUE,TRUE,TRUE,TRUE];
    LockerAccessCode : ARRAY[1..10] OF INT := [1234,5678,9876,4321,6543,7890,3456,8765,2345,6789];
    bInitialized : BOOL := FALSE;
END_VAR

(* One-time initialization *)
IF NOT bInitialized THEN
    bInitialized := TRUE;
END_IF;

(* Reset output at beginning of each cycle *)
LockerOpen := FALSE;

(* Access control logic *)
IF (LockerNumber >= 1) AND (LockerNumber <= 10) THEN
    IF AccessCode = LockerAccessCode[LockerNumber] THEN
        IF LockerStatus[LockerNumber] THEN
            LockerOpen := TRUE;
            LockerStatus[LockerNumber] := FALSE;
        END_IF;
    END_IF;
END_IF;

END_FUNCTION_BLOCK

(* ---- med_89.st ---- *)
FUNCTION_BLOCK SoilTestingDeviceControl
VAR_INPUT
    StartButton : BOOL;           (* Input for starting the testing process *)
    SoilSampleDetected : BOOL;    (* Input for detecting soil sample *)
END_VAR
VAR_OUTPUT
    NutrientPump : BOOL;          (* Output to control nutrient pump *)
    pHAdjustmentPump : BOOL;      (* Output to control pH adjustment pump *)
END_VAR
VAR
    pHSensorValue : REAL;         (* Simulated pH sensor value *)
    NutrientSensorValue : REAL;   (* Simulated nutrient sensor value *)
    TestingStatus : INT;          (* Status: 0=Idle, 1=Testing, 2=Completed *)
    NutrientThreshold : REAL := 0.7;  (* Nutrient level threshold for analysis *)
    pHThreshold : REAL := 6.5;        (* pH level threshold for analysis *)
END_VAR

(* Main state machine logic *)
CASE TestingStatus OF
    0: (* Idle state *)
        (* Initialize sensor values *)
        pHSensorValue := 7.0;
        NutrientSensorValue := 0.5;

        (* Ensure pumps are off in idle state *)
        NutrientPump := FALSE;
        pHAdjustmentPump := FALSE;

        (* Transition to Testing state when StartButton is pressed *)
        IF StartButton THEN
            TestingStatus := 1;
        END_IF;

    1: (* Testing state *)
        (* Activate both pumps during testing *)
        NutrientPump := TRUE;
        pHAdjustmentPump := TRUE;

        (* Update simulated sensor values with limits *)
        NutrientSensorValue := LIMIT(0.5, NutrientSensorValue + 0.1, 0.9);
        pHSensorValue := LIMIT(4.0, pHSensorValue - 0.5, 7.0);

        (* Check for sample detection and threshold conditions *)
        IF SoilSampleDetected THEN
            IF (NutrientSensorValue >= NutrientThreshold) AND (pHSensorValue <= pHThreshold) THEN
                TestingStatus := 2;  (* Transition to Completed state *)
            END_IF;
        END_IF;

    2: (* Completed state *)
        (* Deactivate pumps when testing is complete *)
        NutrientPump := FALSE;
        pHAdjustmentPump := FALSE;

        (* Optionally: Add logic to reset to idle state if needed *)
        (* IF ResetCondition THEN TestingStatus := 0; END_IF *)

END_CASE;

END_FUNCTION_BLOCK

(* ---- med_90.st ---- *)
FUNCTION_BLOCK SushiConveyorControl
VAR_INPUT
    StartButton : BOOL;     (* Input to start the conveyor *)
    StopButton : BOOL;      (* Input to stop the conveyor *)
    EmergencyStop : BOOL;   (* Input for emergency stop *)
END_VAR
VAR_OUTPUT
    ConveyorMotor : BOOL;   (* Output to control the conveyor motor *)
END_VAR
VAR
    BeltRunning : BOOL;     (* Status of the conveyor: Running or Stopped *)
    ConveyorTimer : INT;    (* Timer counter for conveyor rotation *)
    RotationTime : INT := 5; (* Time for one rotation in seconds *)
    PrevStartButton : BOOL; (* Previous state of StartButton for edge detection *)
    PrevStopButton : BOOL;  (* Previous state of StopButton for edge detection *)
END_VAR

(* Initialization *)
BeltRunning := FALSE;
ConveyorMotor := FALSE;
ConveyorTimer := 0;
PrevStartButton := FALSE;
PrevStopButton := FALSE;

(* Emergency Stop - Highest Priority *)
IF EmergencyStop THEN
    ConveyorMotor := FALSE;
    BeltRunning := FALSE;
    ConveyorTimer := 0;
    RETURN;
END_IF;

(* Start/Stop Control with edge detection *)
IF StartButton AND NOT PrevStartButton AND NOT BeltRunning THEN
    (* Rising edge detected on StartButton when conveyor is stopped *)
    ConveyorMotor := TRUE;
    BeltRunning := TRUE;
    ConveyorTimer := 0;
ELSIF StopButton AND NOT PrevStopButton AND BeltRunning THEN
    (* Rising edge detected on StopButton when conveyor is running *)
    ConveyorMotor := FALSE;
    BeltRunning := FALSE;
    ConveyorTimer := 0;
END_IF;

(* Simulated Rotation (Timed On/Off Cycle) *)
IF BeltRunning THEN
    (* Increment timer each scan cycle when running *)
    ConveyorTimer := ConveyorTimer + 1;

    (* Check if timer has reached rotation time *)
    IF ConveyorTimer >= RotationTime THEN
        ConveyorTimer := 0;  (* Reset timer for next cycle *)
        (* For on/off cycle simulation, toggle motor state *)
        ConveyorMotor := NOT ConveyorMotor;
    END_IF;
ELSE
    (* Ensure motor is off when not running *)
    ConveyorMotor := FALSE;
END_IF;

(* Store current button states for next edge detection *)
PrevStartButton := StartButton;
PrevStopButton := StopButton;

END_FUNCTION_BLOCK

(* ---- med_91.st ---- *)
FUNCTION_BLOCK AGVControlSystem
VAR_INPUT
    MaterialRequest : INT; (* New material handling request, positive value indicates valid request *)
END_VAR

VAR_OUTPUT
    AGV1_Ready : BOOL := TRUE; (* AGV 1 ready status *)
    AGV2_Ready : BOOL := TRUE; (* AGV 2 ready status *)
    AGV3_Ready : BOOL := TRUE; (* AGV 3 ready status *)
    QueueStatus : INT := 0; (* Current number of tasks in queue *)
    SystemError : BOOL := FALSE; (* System error flag *)
    ErrorCode : INT := 0; (* Error code: 0=No error, 1=Queue overflow, 2=Invalid request, 3=Position error *)
END_VAR

VAR
    (* Queue management variables *)
    MaterialQueue : ARRAY[1..10] OF INT; (* Material handling request queue *)
    QueueHead : INT := 1; (* Index of first element in queue *)
    QueueTail : INT := 1; (* Index where next element will be inserted *)
    QueueCount : INT := 0; (* Current number of elements in queue *)

    (* AGV status tracking *)
    AGVPosition : ARRAY[1..3] OF INT := [0,0,0]; (* Current position of each AGV *)
    AGVTask : ARRAY[1..3] OF INT := [0,0,0]; (* Current task assigned to each AGV *)
    AGVWorking : ARRAY[1..3] OF BOOL := [FALSE,FALSE,FALSE]; (* Working status of each AGV *)

    (* Internal flags and counters *)
    TaskInProgress : BOOL := FALSE; (* Flag indicating if any AGV is working *)
    i : INT; (* Loop counter *)
    TempRequest : INT; (* Temporary request storage *)
END_VAR

(* Initialize error states *)
SystemError := FALSE;
ErrorCode := 0;

(* 1. Queue Management - Process new material requests *)
IF MaterialRequest > 0 THEN
    (* Validate request *)
    IF MaterialRequest <= 0 THEN
        SystemError := TRUE;
        ErrorCode := 2; (* Invalid request *)
    ELSIF QueueCount >= 10 THEN
        SystemError := TRUE;
        ErrorCode := 1; (* Queue overflow *)
    ELSE
        (* Add request to queue - atomic operation *)
        MaterialQueue[QueueTail] := MaterialRequest;

        (* Update queue tail with wrap-around *)
        QueueTail := QueueTail + 1;
        IF QueueTail > 10 THEN
            QueueTail := 1;
        END_IF;

        (* Update queue count *)
        QueueCount := QueueCount + 1;
    END_IF;
END_IF;

(* 2. AGV Status Management - Update AGV ready status *)
AGV1_Ready := NOT AGVWorking[1];
AGV2_Ready := NOT AGVWorking[2];
AGV3_Ready := NOT AGVWorking[3];

(* 3. Task Execution Simulation - Simulate AGV movement and task completion *)
FOR i := 1 TO 3 DO
    IF AGVWorking[i] THEN
        (* Simulate AGV movement - increment position *)
        AGVPosition[i] := AGVPosition[i] + 1;

        (* Simulate task completion at position 100 *)
        IF AGVPosition[i] >= 100 THEN
            (* Task completed - reset AGV state *)
            AGVWorking[i] := FALSE;
            AGVTask[i] := 0;
            AGVPosition[i] := 0; (* Return to start position *)
        END_IF;
    END_IF;
END_FOR;

(* 4. Check if any task is in progress *)
TaskInProgress := FALSE;
FOR i := 1 TO 3 DO
    IF AGVWorking[i] THEN
        TaskInProgress := TRUE;
        EXIT;
    END_IF;
END_FOR;

(* 5. Priority-based Task Assignment *)
(* Only assign tasks if queue is not empty and no task is currently being assigned *)
IF (QueueCount > 0) AND (NOT TaskInProgress) THEN
    (* Priority order: AGV1 > AGV2 > AGV3 *)
    IF AGV1_Ready THEN
        (* Assign task to AGV1 *)
        AGVTask[1] := MaterialQueue[QueueHead];
        AGVWorking[1] := TRUE;

        (* Remove task from queue - atomic operation *)
        QueueHead := QueueHead + 1;
        IF QueueHead > 10 THEN
            QueueHead := 1;
        END_IF;
        QueueCount := QueueCount - 1;

    ELSIF AGV2_Ready THEN
        (* Assign task to AGV2 *)
        AGVTask[2] := MaterialQueue[QueueHead];
        AGVWorking[2] := TRUE;

        (* Remove task from queue *)
        QueueHead := QueueHead + 1;
        IF QueueHead > 10 THEN
            QueueHead := 1;
        END_IF;
        QueueCount := QueueCount - 1;

    ELSIF AGV3_Ready THEN
        (* Assign task to AGV3 *)
        AGVTask[3] := MaterialQueue[QueueHead];
        AGVWorking[3] := TRUE;

        (* Remove task from queue *)
        QueueHead := QueueHead + 1;
        IF QueueHead > 10 THEN
            QueueHead := 1;
        END_IF;
        QueueCount := QueueCount - 1;
    END_IF;
END_IF;

(* 6. Safety Constraints - Ensure non-negative positions *)
FOR i := 1 TO 3 DO
    IF AGVPosition[i] < 0 THEN
        AGVPosition[i] := 0;
        SystemError := TRUE;
        ErrorCode := 3; (* Position error *)
    END_IF;
END_FOR;

(* 7. Queue boundary validation *)
IF QueueCount < 0 THEN
    QueueCount := 0;
ELSIF QueueCount > 10 THEN
    QueueCount := 10;
    SystemError := TRUE;
    ErrorCode := 1; (* Queue overflow *)
END_IF;

IF QueueHead < 1 THEN
    QueueHead := 1;
ELSIF QueueHead > 10 THEN
    QueueHead := 10;
END_IF;

IF QueueTail < 1 THEN
    QueueTail := 1;
ELSIF QueueTail > 10 THEN
    QueueTail := 10;
END_IF;

(* 8. Output queue status *)
QueueStatus := QueueCount;

(* 9. System state validation - ensure consistency *)
IF (QueueCount = 0) AND (NOT AGVWorking[1]) AND (NOT AGVWorking[2]) AND (NOT AGVWorking[3]) THEN
    (* System in idle state - all resources released *)
    (* Additional cleanup if needed *)
END_IF;

END_FUNCTION_BLOCK
